// TIA Portal project "JAVA" (V11)

(* hardware
DEVICE "S7300/ET200 station_1"  SIMATIC 300-Station
   slot 0: "Perfil soporte_0"  Rail  6ES7 390-1***0-0AA0
   slot 2: "PLC_1"  CPU 313C-2 DP  6ES7 313-6CF03-0AB0  V2.6
      slot 0: "Interfaz MPI_1"  MPI
      slot 1: "Interfaz DP_1"  DP
      slot 2: "DI16/DO16_1"  DI16/DO16
      slot 4: "Contaje_1"  Counter
*)

// ===== PLC "PLC_1"  CPU 313C-2 DP =====

VAR_GLOBAL   // PLC tag table "Tabla de variables estándar"
   "Tag_1" AT %E0.0 : Bool;
   "Tag_2" AT %A0.0 : Bool;
   "Tag_3" AT %E0.1 : Bool;
   "Tag_4" AT %E0.2 : Bool;
   "Tag_5" AT %A0.1 : Bool;
END_VAR

DATA_BLOCK "INICIO_DB"   // DB1
{ S7_Optimized_Access := 'FALSE' }
VERSION : 0.1
// stored: InstanceOfName INICIO
"INICIO"
BEGIN
END_DATA_BLOCK

FUNCTION_BLOCK "INICIO"   // FB1, SCL
{ S7_Optimized_Access := 'FALSE' }
VERSION : 0.1
   VAR_INPUT
      MARCHA : Bool;
      PARO : Bool;
      PULSO : Bool;
   END_VAR
   VAR_OUTPUT
      MOTOR : Bool;
      LED : Bool;
   END_VAR
BEGIN
   IF #MARCHA THEN
     #MOTOR := TRUE;
   END_IF;
   IF #PARO THEN
     #MOTOR := FALSE;
   END_IF;
   IF #PULSO THEN
     #LED := TRUE;
   ELSE
     #LED := FALSE ;
     END_IF ;
END_FUNCTION_BLOCK

ORGANIZATION_BLOCK "Main"   // OB1, LAD
TITLE = "Main Program Sweep (Cycle)"
{ S7_Optimized_Access := 'FALSE' }
VERSION : 0.1
   VAR_TEMP
      OB1_EV_CLASS : Byte;   // Bits 0-3 = 1 (Coming event), Bits 4-7 = 1 (Event class 1)
      OB1_SCAN_1 : Byte;   // 1 (Cold restart scan 1 of OB 1), 3 (Scan 2-n of OB 1)
      OB1_PRIORITY : Byte;   // Priority of OB Execution
      OB1_OB_NUMBR : Byte;   // 1 (Organization block 1, OB1)
      OB1_RESERVED_1 : Byte;   // Reserved for system
      OB1_RESERVED_2 : Byte;   // Reserved for system
      OB1_PREV_CYCLE : Int;   // Cycle time of previous OB1 scan (milliseconds)
      OB1_MIN_CYCLE : Int;   // Minimum cycle time of OB1 (milliseconds)
      OB1_MAX_CYCLE : Int;   // Maximum cycle time of OB1 (milliseconds)
      OB1_DATE_TIME : Date_And_Time;   // Date and time OB1 started
   END_VAR
BEGIN

REGION Network 1
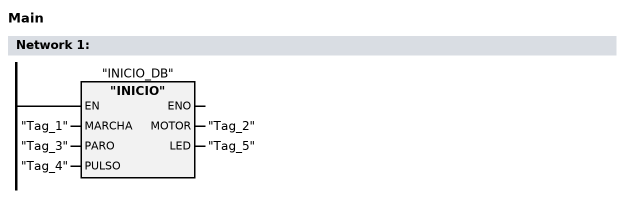
   RUNG wire#powerrail
      "INICIO_DB"(MARCHA := "Tag_1", PARO := "Tag_3", PULSO := "Tag_4", MOTOR => "Tag_2", LED => "Tag_5")
   END_RUNG
   // the same network as SCL:
   "INICIO_DB"(MARCHA := "Tag_1", PARO := "Tag_3", PULSO := "Tag_4", MOTOR => "Tag_2", LED => "Tag_5");   // "INICIO"
END_REGION
END_ORGANIZATION_BLOCK